Staubli VAL3: mnuEnterIPVals.pgx

program mnuEnterIPVals()
  local bool LbBackup
  local num nKey
begin
  //
  //header begin
  //
  //  pgm mnuEnterIPVals()
  // this program allows user to set global Interaction Point values
  //
  //  incoming parms: none
  //  outgoing parms: none
  //
  //  called from mnuTeachIP()
  //
  //  Added for Release 2: KN
  //
  //header end
  //
  // set up display
  LbBackup=false
  do
    // nIdxEnterIP=341
    call displayMessage7(nIdxEnterIP,nKey)
    // verify selection
    switch nKey
      // ESC key aborts immediately
      case 255
        return
      break
      // menu = Direct Entry TCP values, F1 button = IP-X value
      case 271
        gotoxy(18,3)
        if nIPNumber==-1
          get(fIPoriginal.trsf.x)
        elseIf nIPNumber==0
          get(fIP1.trsf.x)
        else
          get(fIP2.trsf.x)
        endIf
      break
      // menu = Direct Entry TCP values,  F2 Button = IP-Y value
      case 272
        gotoxy(18,4)
        if nIPNumber==-1
          get(fIPoriginal.trsf.y)
        elseIf nIPNumber==0
          get(fIP1.trsf.y)
        else
          get(fIP2.trsf.y)
        endIf
      break
      // menu = Direct Entry TCP Values,  F3 Button = IP-Z value
      case 273
        gotoxy(18,5)
        if nIPNumber==-1
          get(fIPoriginal.trsf.z)
        elseIf nIPNumber==0
          get(fIP1.trsf.z)
        else
          get(fIP2.trsf.z)
        endIf
      break
      // menu = Direct Entry TCP values, F4 Button = IP-RX value
      case 274
        gotoxy(18,6)
        if nIPNumber==-1
          get(fIPoriginal.trsf.rx)
        elseIf nIPNumber==0
          get(fIP1.trsf.rx)
        else
          get(fIP2.trsf.rx)
        endIf
      break
      // menu = Direct Entry TCP Values, F5 Button = IP-RY value
      case 275
        gotoxy(18,7)
        if nIPNumber==-1
          get(fIPoriginal.trsf.ry)
        elseIf nIPNumber==0
          get(fIP1.trsf.ry)
        else
          get(fIP2.trsf.ry)
        endIf
      break
      // menu = Direct Entry TCP Values, F6 Button = IP-RZ value
      case 276
        gotoxy(18,8)
        if nIPNumber==-1
          get(fIPoriginal.trsf.rz)
        elseIf nIPNumber==0
          get(fIP1.trsf.rz)
        else
          get(fIP2.trsf.rz)
        endIf
      break
      // menu = Main Menu:  F8 Button, Save updated TCP values & return to pgm mnuTeachIP()
      case 278
        LbBackup=true
        libSave()
      break
      // ALL OTHER CHOICES
      default
        popUpMsg("EnterIPVals:  BAD SELECTION...Press OK")
      break
    endSwitch
  until (false or (LbBackup==true))
end
